// TIA Portal V17 export
// export: Created 2022-07-20T07:01:25.3960544Z, ExportSetting WithDefaults, DisplayName Totally Integrated Automation Portal, DisplayVersion V17, DisplayName TIA Portal Openness, DisplayVersion V17, DisplayName TIA Portal Version Control Interface, DisplayVersion V17, DisplayName SINAMICS Startdrive Advanced, DisplayVersion V17, DisplayName SINAMICS Startdrive G130, G150, S120, S150, SINAMICS MV, S210, DisplayVersion V17, DisplayName SINAMICS Startdrive G110M, G120, G120C, G120D, G120P, G115D, DisplayVersion V17, DisplayName STEP 7 Professional, DisplayVersion V17, DisplayName STEP 7 Safety, DisplayVersion V17, DisplayName WinCC Advanced, DisplayVersion V17
FUNCTION_BLOCK "FB10230_LAM_LexiumDriver"   // FB10230, LAD
{ S7_Optimized_Access := 'TRUE' }
AUTHOR : Schneider_Electric
FAMILY : Lexium_MDrive
VERSION : 1.0
// stored: AutoNumber false, IsIECCheckEnabled false, IsRetainMemResEnabled false, MemoryReserve 100, SetENOAutomatically false, UDAEnableTagReadback false
   VAR_INPUT
      Drive_In : "TLexium_MDrv_Drv2Plc";
      UseInputsOutputs : Bool;
      Move_Type : DInt;
      Home_Type : SInt := 1;
      Position : DInt;
      Speed : DWord := 20000;
      Jog_Speed : DInt := 75000;
      Accel_Rate : DWord := 10000;
      Decel_Rate : DWord := 10000;
      Initial_Vel : DWord := 1000;
      Hold_Current : SInt := 5;
      Run_Current : SInt := 25;
      MicrostepValue : DInt := 256;
      Enable : Bool;
      Start : Bool;
      Stop : Bool;
      Jog_Fwd : Bool;
      Jog_Rev : Bool;
      Acknowledge : Bool;
      Home : Bool;
      Zero_Home_Pos : Bool := false;
      Out1_Set : Bool;
      Out2_Set : Bool;
      Out3_Set : Bool;
   END_VAR
   VAR_OUTPUT
      Drive_Out : "TLexium_MDrv_Plc2Drv";
      Pos_Fdbk : DInt;
      Error_Code : UInt;
      DN : Bool;
      ER : Bool;
      IP : Bool;
      In1 : Bool;
      In2 : Bool;
      In3 : Bool;
      In4 : Bool;
   END_VAR
   VAR
      Jog_Perm : Bool;
      Jog_Fwd_Req : Bool;
      Jog_Rev_Req : Bool;
      Stop_Act : Bool;
      Abs_Act : Bool;
      Rel_Act : Bool;
      HM_Act : Bool;
      Start_OS : Bool;
      MV_Stop_OS : Bool;
      Set_Pos_Zero : Bool;
      Slew_Rate : DInt;
      Slew_Rate_Prev : DInt;
      MicrostepValue_Prev : DInt;
      SetAccTmr { S7_SetPoint := 'True'} : TOF_TIME;
      SetDecTmr { S7_SetPoint := 'True'} : TOF_TIME;
      SetTSTmr { S7_SetPoint := 'True'} : TOF_TIME;
      SetVITmr { S7_SetPoint := 'True'} : TOF_TIME;
      SetVMTmr { S7_SetPoint := 'True'} : TOF_TIME;
      SetHCTmr { S7_SetPoint := 'True'} : TOF_TIME;
      SetRCTmr { S7_SetPoint := 'True'} : TOF_TIME;
      SetTQTmr { S7_SetPoint := 'True'} : TOF_TIME;
      SetSLTmr { S7_SetPoint := 'True'} : TOF_TIME;
      ABS_Tmr { S7_SetPoint := 'True'} : TOF_TIME;
      REL_Tmr { S7_SetPoint := 'True'} : TOF_TIME;
      HM_Tmr { S7_SetPoint := 'True'} : TOF_TIME;
      MS_Tmr { S7_SetPoint := 'True'} : TOF_TIME;
      SetZero_Tmr { S7_SetPoint := 'True'} : TOF_TIME;
      ClrErr_Tmr { S7_SetPoint := 'True'} : TOF_TIME;
      Stop_Dly_Tmr { S7_SetPoint := 'True'} : TON_TIME;
      ACC_PMem : Bool;
      DEC_PMem : Bool;
      TS_PMem : Bool;
      VI_PMem : Bool;
      VM_PMem : Bool;
      HC_PMem : Bool;
      RC_PMem : Bool;
      TQ_PMem : Bool;
      SL_PMem : Bool;
      MS_Pmem : Bool;
      Start_PMem : Bool;
      MV_NMem : Bool;
      ABS_PMem : Bool;
      REL_PMem : Bool;
      HM_PMem : Bool;
      Set_Zero_PMem : Bool;
      ClrErr_PMem : Bool;
      AckErr_Pmem : Bool;
      Stop_PMem : Bool;
      MV_Stop_Tmr { S7_SetPoint := 'True'} : TON_TIME;
      IS_PMem { S7_SetPoint := 'True'} : Bool;
      FB10232_Lam_WriteISMessages_Instance { S7_SetPoint := 'True'} : "FB10232_LAM_WriteISMessages";
   END_VAR
   VAR_TEMP
      Inputs : SInt;
      Hold_Cur_SP : SInt;
      Run_Cur_SP : SInt;
      Torque_SP : SInt;
      Move_Type_Loc : DInt;
      Home_Type_Loc : SInt;
      Position_SP : DInt;
      _SetAccTmr_ET : Time;
      _SetDecTmr_ET : Time;
      _SetTSTmr_ET : Time;
      _SetVITmr_ET : Time;
      _SetVMTmr_ET : Time;
      _SetHCTmr_ET : Time;
      _SetRCTmr_ET : Time;
      _SetTQTmr_ET : Time;
      _SetSLTmr_ET : Time;
      _Abs_Tmr_ET : Time;
      _Rel_Tmr_ET : Time;
      _HM_Tmr_ET : Time;
      _SetZero_Tmr_ET : Time;
      _Stop_Dly_Tmr_ET : Time;
      _ClrErr_Tmr_ET : Time;
      Outputs : SInt;
   END_VAR
   // Drive_Out.AS := 2;   // 2 = Mode hybride
   VAR_TEMP   // added for the SCL form of the ladder/FBD networks
      _w1 : Bool;
      _w2 : Bool;
      _w3 : Bool;
      _w4 : Bool;
   END_VAR
BEGIN

REGION Network 1: States of Inputs In1, 2, 3, 4
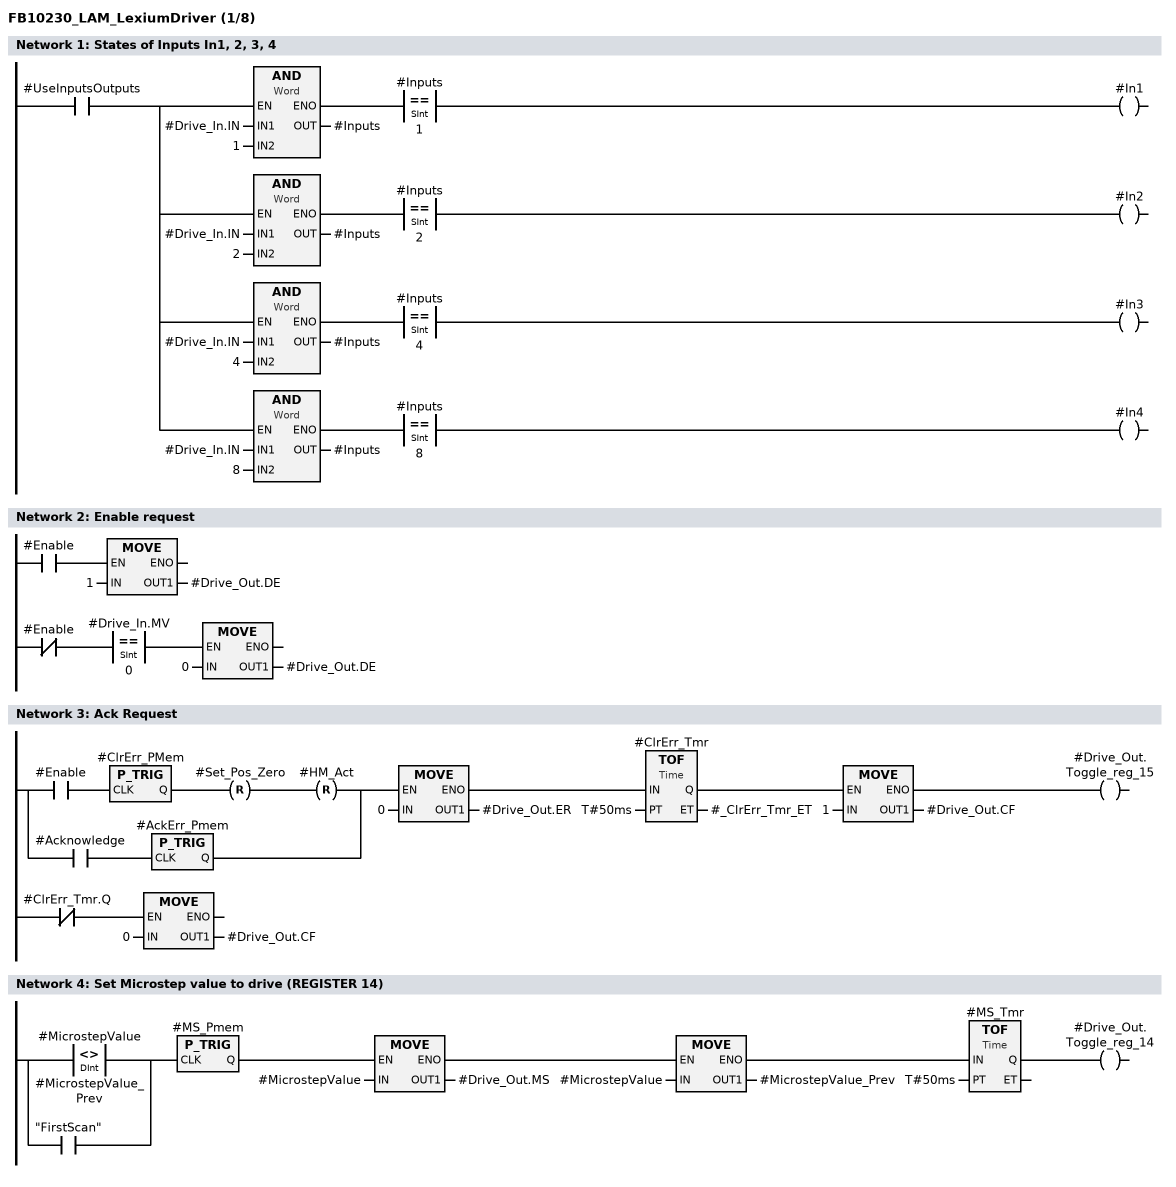
   RUNG wire#powerrail
      Contact( #UseInputsOutputs )
      wire#w1
      { S7_Templates := "SrcType := Word" } And(in1 := #Drive_In.IN, in2 := 1, out => #Inputs)
      { S7_Templates := "SrcType := SInt" } EQ_Contact(in1 := #Inputs, in2 := 1)
      Coil( #In1 )
   END_RUNG
   RUNG wire#w1
      { S7_Templates := "SrcType := Word" } And(in1 := #Drive_In.IN, in2 := 2, out => #Inputs)
      { S7_Templates := "SrcType := SInt" } EQ_Contact(in1 := #Inputs, in2 := 2)
      Coil( #In2 )
   END_RUNG
   RUNG wire#w1
      { S7_Templates := "SrcType := Word" } And(in1 := #Drive_In.IN, in2 := 4, out => #Inputs)
      { S7_Templates := "SrcType := SInt" } EQ_Contact(in1 := #Inputs, in2 := 4)
      Coil( #In3 )
   END_RUNG
   RUNG wire#w1
      { S7_Templates := "SrcType := Word" } And(in1 := #Drive_In.IN, in2 := 8, out => #Inputs)
      { S7_Templates := "SrcType := SInt" } EQ_Contact(in1 := #Inputs, in2 := 8)
      Coil( #In4 )
   END_RUNG
   // the same network as SCL:
   IF #UseInputsOutputs THEN #Inputs := #Drive_In.IN AND 1; END_IF;
   #In1 := #UseInputsOutputs AND (#Inputs = 1);
   IF #UseInputsOutputs THEN #Inputs := #Drive_In.IN AND 2; END_IF;
   #In2 := #UseInputsOutputs AND (#Inputs = 2);
   IF #UseInputsOutputs THEN #Inputs := #Drive_In.IN AND 4; END_IF;
   #In3 := #UseInputsOutputs AND (#Inputs = 4);
   IF #UseInputsOutputs THEN #Inputs := #Drive_In.IN AND 8; END_IF;
   #In4 := #UseInputsOutputs AND (#Inputs = 8);
END_REGION

REGION Network 2: Enable request
   RUNG wire#powerrail
      Contact( #Enable )
      Move(in := 1, out1 => #Drive_Out.DE)
   END_RUNG
   RUNG wire#powerrail
      I_Contact( #Enable )
      { S7_Templates := "SrcType := SInt" } EQ_Contact(in1 := #Drive_In.MV, in2 := 0)
      Move(in := 0, out1 => #Drive_Out.DE)
   END_RUNG
   // the same network as SCL:
   IF #Enable THEN #Drive_Out.DE := 1; END_IF;
   IF NOT #Enable AND (#Drive_In.MV = 0) THEN #Drive_Out.DE := 0; END_IF;
END_REGION

REGION Network 3: Ack Request
   RUNG wire#powerrail
      Contact( #Enable )
      P_Trig( #ClrErr_PMem )
      R_Coil( #Set_Pos_Zero )
      R_Coil( #HM_Act )
      wire#w1
      Move(in := 0, out1 => #Drive_Out.ER)
      { S7_Templates := "time_type := Time" } #ClrErr_Tmr.TOF(pt := T#50ms, et => #_ClrErr_Tmr_ET)
      Move(in := 1, out1 => #Drive_Out.CF)
      Coil( #Drive_Out.Toggle_reg_15 )
   END_RUNG
   RUNG wire#powerrail
      Contact( #Acknowledge )
      P_Trig( #AckErr_Pmem )
   END_RUNG wire#w1
   RUNG wire#powerrail
      I_Contact( #ClrErr_Tmr.Q )
      Move(in := 0, out1 => #Drive_Out.CF)
   END_RUNG
   // the same network as SCL:
   #_w1 := #Enable AND NOT #ClrErr_PMem;   // rising edge
   #ClrErr_PMem := #Enable;
   IF #_w1 THEN
       #Set_Pos_Zero := FALSE;
       #HM_Act := FALSE;
   END_IF;
   #_w2 := #Acknowledge AND NOT #AckErr_Pmem;   // rising edge
   #AckErr_Pmem := #Acknowledge;
   #_w3 := #_w1 OR #_w2;
   IF #_w3 THEN #Drive_Out.ER := 0; END_IF;
   #ClrErr_Tmr(IN := #_w3, PT := T#50ms, ET => #_ClrErr_Tmr_ET);   // TOF
   IF #ClrErr_Tmr.Q THEN #Drive_Out.CF := 1; END_IF;
   #Drive_Out.Toggle_reg_15 := #ClrErr_Tmr.Q;
   IF NOT #ClrErr_Tmr.Q THEN #Drive_Out.CF := 0; END_IF;
END_REGION

REGION Network 4: Set Microstep value to drive (REGISTER 14)
   RUNG wire#powerrail
      { S7_Templates := "SrcType := DInt" } NE_Contact(in1 := #MicrostepValue, in2 := #MicrostepValue_Prev)
      wire#w1
      P_Trig( #MS_Pmem )
      Move(in := #MicrostepValue, out1 => #Drive_Out.MS)
      Move(in := #MicrostepValue, out1 => #MicrostepValue_Prev)
      { S7_Templates := "time_type := Time" } #MS_Tmr.TOF(pt := T#50ms, et =>)
      Coil( #Drive_Out.Toggle_reg_14 )
   END_RUNG
   RUNG wire#powerrail
      Contact( "FirstScan" )
   END_RUNG wire#w1
   // the same network as SCL:
   #_w1 := (#MicrostepValue <> #MicrostepValue_Prev) OR "FirstScan";
   #_w2 := #_w1 AND NOT #MS_Pmem;   // rising edge
   #MS_Pmem := #_w1;
   IF #_w2 THEN
       #Drive_Out.MS := #MicrostepValue;
       #MicrostepValue_Prev := #MicrostepValue;
   END_IF;
   #MS_Tmr(IN := #_w2, PT := T#50ms);   // TOF
   #Drive_Out.Toggle_reg_14 := #MS_Tmr.Q;
END_REGION

REGION Network 5: Hold Current limits
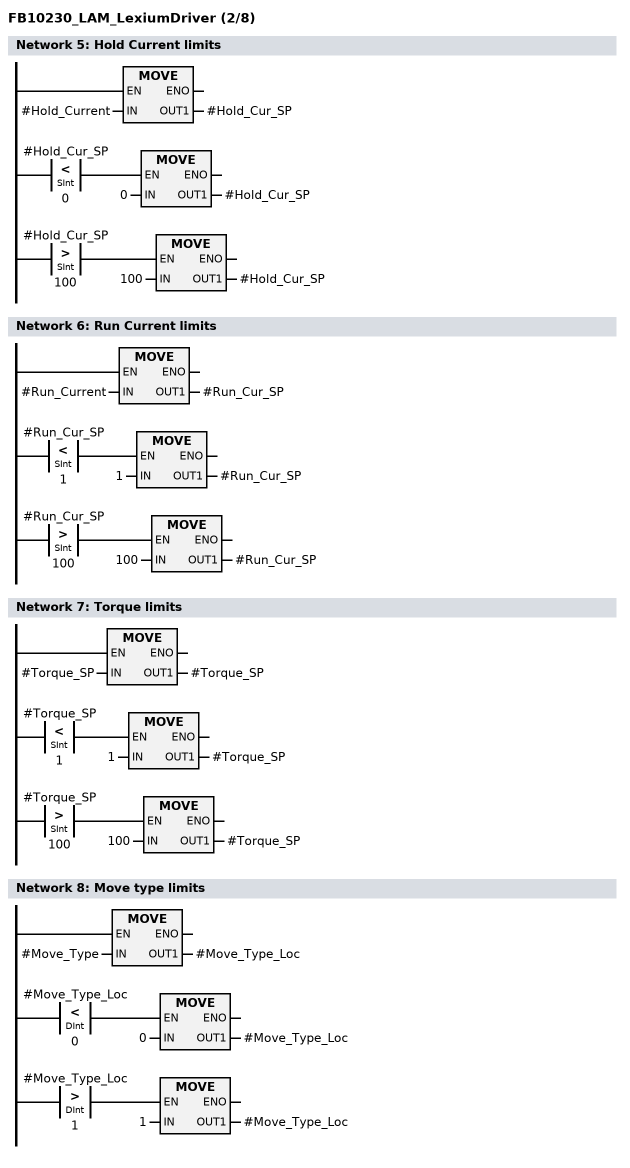
   RUNG wire#powerrail
      Move(in := #Hold_Current, out1 => #Hold_Cur_SP)
   END_RUNG
   RUNG wire#powerrail
      { S7_Templates := "SrcType := SInt" } LT_Contact(in1 := #Hold_Cur_SP, in2 := 0)
      Move(in := 0, out1 => #Hold_Cur_SP)
   END_RUNG
   RUNG wire#powerrail
      { S7_Templates := "SrcType := SInt" } GT_Contact(in1 := #Hold_Cur_SP, in2 := 100)
      Move(in := 100, out1 => #Hold_Cur_SP)
   END_RUNG
   // the same network as SCL:
   #Hold_Cur_SP := #Hold_Current;
   IF #Hold_Cur_SP < 0 THEN #Hold_Cur_SP := 0; END_IF;
   IF #Hold_Cur_SP > 100 THEN #Hold_Cur_SP := 100; END_IF;
END_REGION

REGION Network 6: Run Current limits
   RUNG wire#powerrail
      Move(in := #Run_Current, out1 => #Run_Cur_SP)
   END_RUNG
   RUNG wire#powerrail
      { S7_Templates := "SrcType := SInt" } LT_Contact(in1 := #Run_Cur_SP, in2 := 1)
      Move(in := 1, out1 => #Run_Cur_SP)
   END_RUNG
   RUNG wire#powerrail
      { S7_Templates := "SrcType := SInt" } GT_Contact(in1 := #Run_Cur_SP, in2 := 100)
      Move(in := 100, out1 => #Run_Cur_SP)
   END_RUNG
   // the same network as SCL:
   #Run_Cur_SP := #Run_Current;
   IF #Run_Cur_SP < 1 THEN #Run_Cur_SP := 1; END_IF;
   IF #Run_Cur_SP > 100 THEN #Run_Cur_SP := 100; END_IF;
END_REGION

REGION Network 7: Torque limits
   RUNG wire#powerrail
      Move(in := #Torque_SP, out1 => #Torque_SP)
   END_RUNG
   RUNG wire#powerrail
      { S7_Templates := "SrcType := SInt" } LT_Contact(in1 := #Torque_SP, in2 := 1)
      Move(in := 1, out1 => #Torque_SP)
   END_RUNG
   RUNG wire#powerrail
      { S7_Templates := "SrcType := SInt" } GT_Contact(in1 := #Torque_SP, in2 := 100)
      Move(in := 100, out1 => #Torque_SP)
   END_RUNG
   // the same network as SCL:
   #Torque_SP := #Torque_SP;
   IF #Torque_SP < 1 THEN #Torque_SP := 1; END_IF;
   IF #Torque_SP > 100 THEN #Torque_SP := 100; END_IF;
END_REGION

REGION Network 8: Move type limits
   RUNG wire#powerrail
      Move(in := #Move_Type, out1 => #Move_Type_Loc)
   END_RUNG
   RUNG wire#powerrail
      { S7_Templates := "SrcType := DInt" } LT_Contact(in1 := #Move_Type_Loc, in2 := 0)
      Move(in := 0, out1 => #Move_Type_Loc)
   END_RUNG
   RUNG wire#powerrail
      { S7_Templates := "SrcType := DInt" } GT_Contact(in1 := #Move_Type_Loc, in2 := 1)
      Move(in := 1, out1 => #Move_Type_Loc)
   END_RUNG
   // the same network as SCL:
   #Move_Type_Loc := #Move_Type;
   IF #Move_Type_Loc < 0 THEN #Move_Type_Loc := 0; END_IF;
   IF #Move_Type_Loc > 1 THEN #Move_Type_Loc := 1; END_IF;
END_REGION

REGION Network 9: Home type limits
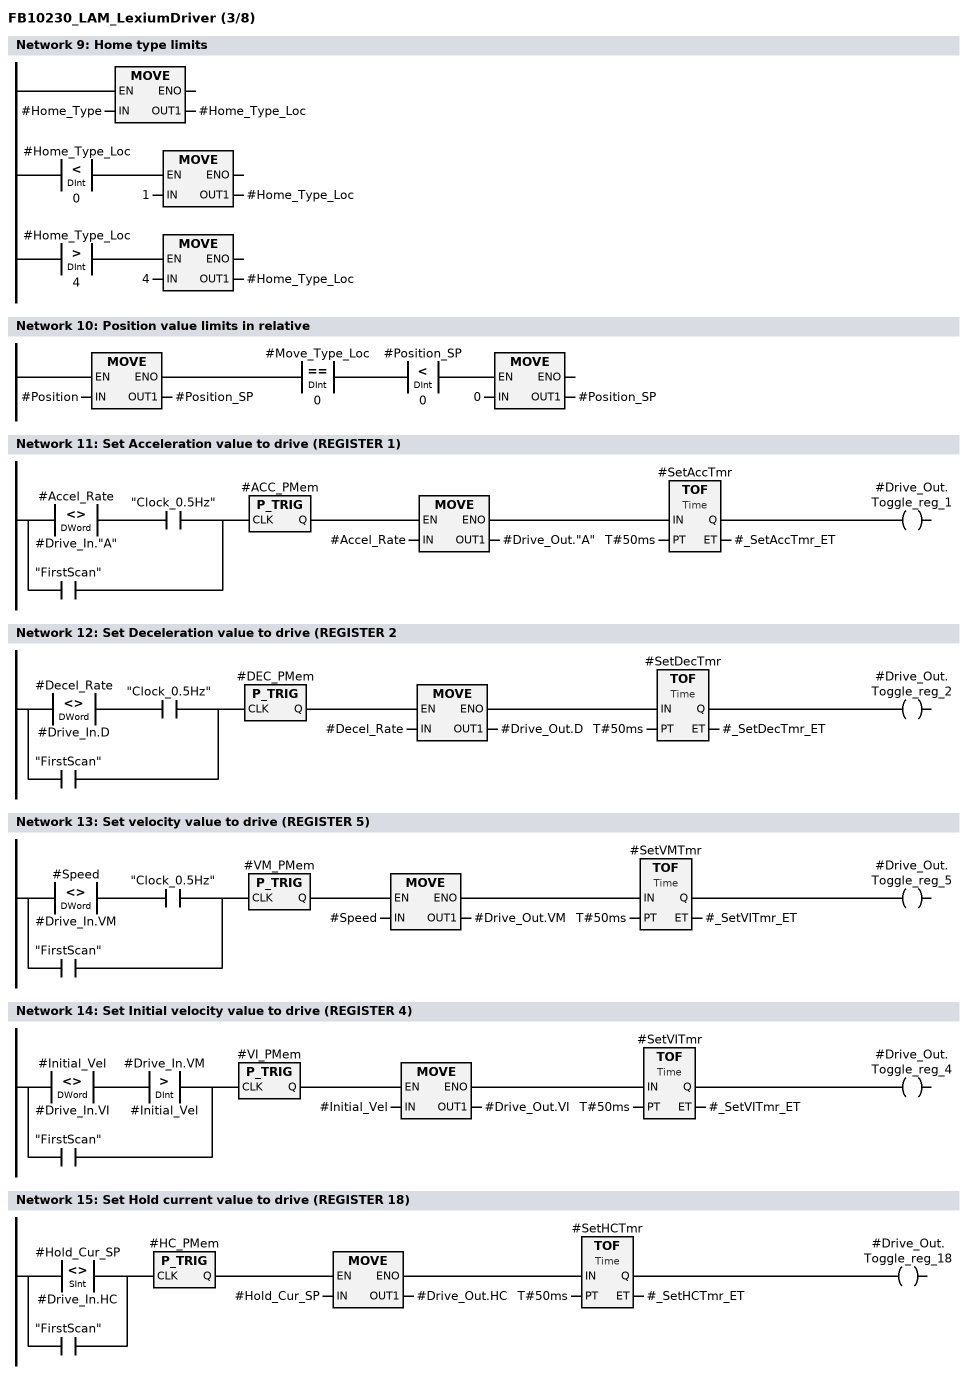
   RUNG wire#powerrail
      Move(in := #Home_Type, out1 => #Home_Type_Loc)
   END_RUNG
   RUNG wire#powerrail
      { S7_Templates := "SrcType := DInt" } LT_Contact(in1 := #Home_Type_Loc, in2 := 0)
      Move(in := 1, out1 => #Home_Type_Loc)
   END_RUNG
   RUNG wire#powerrail
      { S7_Templates := "SrcType := DInt" } GT_Contact(in1 := #Home_Type_Loc, in2 := 4)
      Move(in := 4, out1 => #Home_Type_Loc)
   END_RUNG
   // the same network as SCL:
   #Home_Type_Loc := #Home_Type;
   IF #Home_Type_Loc < 0 THEN #Home_Type_Loc := 1; END_IF;
   IF #Home_Type_Loc > 4 THEN #Home_Type_Loc := 4; END_IF;
END_REGION

REGION Network 10: Position value limits in relative
   RUNG wire#powerrail
      Move(in := #Position, out1 => #Position_SP)
      { S7_Templates := "SrcType := DInt" } EQ_Contact(in1 := #Move_Type_Loc, in2 := 0)
      { S7_Templates := "SrcType := DInt" } LT_Contact(in1 := #Position_SP, in2 := 0)
      Move(in := 0, out1 => #Position_SP)
   END_RUNG
   // the same network as SCL:
   #Position_SP := #Position;
   IF (#Move_Type_Loc = 0) AND (#Position_SP < 0) THEN #Position_SP := 0; END_IF;
END_REGION

REGION Network 11: Set Acceleration value to drive (REGISTER 1)
   RUNG wire#powerrail
      { S7_Templates := "SrcType := DWord" } NE_Contact(in1 := #Accel_Rate, in2 := #Drive_In."A")
      Contact( "Clock_0.5Hz" )
      wire#w1
      P_Trig( #ACC_PMem )
      Move(in := #Accel_Rate, out1 => #Drive_Out."A")
      { S7_Templates := "time_type := Time" } #SetAccTmr.TOF(pt := T#50ms, et => #_SetAccTmr_ET)
      Coil( #Drive_Out.Toggle_reg_1 )
   END_RUNG
   RUNG wire#powerrail
      Contact( "FirstScan" )
   END_RUNG wire#w1
   // the same network as SCL:
   #_w1 := ((#Accel_Rate <> #Drive_In."A") AND "Clock_0.5Hz") OR "FirstScan";
   #_w2 := #_w1 AND NOT #ACC_PMem;   // rising edge
   #ACC_PMem := #_w1;
   IF #_w2 THEN #Drive_Out."A" := #Accel_Rate; END_IF;
   #SetAccTmr(IN := #_w2, PT := T#50ms, ET => #_SetAccTmr_ET);   // TOF
   #Drive_Out.Toggle_reg_1 := #SetAccTmr.Q;
END_REGION

REGION Network 12: Set Deceleration value to drive (REGISTER 2
   RUNG wire#powerrail
      { S7_Templates := "SrcType := DWord" } NE_Contact(in1 := #Decel_Rate, in2 := #Drive_In.D)
      Contact( "Clock_0.5Hz" )
      wire#w1
      P_Trig( #DEC_PMem )
      Move(in := #Decel_Rate, out1 => #Drive_Out.D)
      { S7_Templates := "time_type := Time" } #SetDecTmr.TOF(pt := T#50ms, et => #_SetDecTmr_ET)
      Coil( #Drive_Out.Toggle_reg_2 )
   END_RUNG
   RUNG wire#powerrail
      Contact( "FirstScan" )
   END_RUNG wire#w1
   // the same network as SCL:
   #_w1 := ((#Decel_Rate <> #Drive_In.D) AND "Clock_0.5Hz") OR "FirstScan";
   #_w2 := #_w1 AND NOT #DEC_PMem;   // rising edge
   #DEC_PMem := #_w1;
   IF #_w2 THEN #Drive_Out.D := #Decel_Rate; END_IF;
   #SetDecTmr(IN := #_w2, PT := T#50ms, ET => #_SetDecTmr_ET);   // TOF
   #Drive_Out.Toggle_reg_2 := #SetDecTmr.Q;
END_REGION

REGION Network 13: Set velocity value to drive (REGISTER 5)
   RUNG wire#powerrail
      { S7_Templates := "SrcType := DWord" } NE_Contact(in1 := #Speed, in2 := #Drive_In.VM)
      Contact( "Clock_0.5Hz" )
      wire#w1
      P_Trig( #VM_PMem )
      Move(in := #Speed, out1 => #Drive_Out.VM)
      { S7_Templates := "time_type := Time" } #SetVMTmr.TOF(pt := T#50ms, et => #_SetVITmr_ET)
      Coil( #Drive_Out.Toggle_reg_5 )
   END_RUNG
   RUNG wire#powerrail
      Contact( "FirstScan" )
   END_RUNG wire#w1
   // the same network as SCL:
   #_w1 := ((#Speed <> #Drive_In.VM) AND "Clock_0.5Hz") OR "FirstScan";
   #_w2 := #_w1 AND NOT #VM_PMem;   // rising edge
   #VM_PMem := #_w1;
   IF #_w2 THEN #Drive_Out.VM := #Speed; END_IF;
   #SetVMTmr(IN := #_w2, PT := T#50ms, ET => #_SetVITmr_ET);   // TOF
   #Drive_Out.Toggle_reg_5 := #SetVMTmr.Q;
END_REGION

REGION Network 14: Set Initial velocity value to drive (REGISTER 4)
   RUNG wire#powerrail
      { S7_Templates := "SrcType := DWord" } NE_Contact(in1 := #Initial_Vel, in2 := #Drive_In.VI)
      { S7_Templates := "SrcType := DInt" } GT_Contact(in1 := #Drive_In.VM, in2 := #Initial_Vel)
      wire#w1
      P_Trig( #VI_PMem )
      Move(in := #Initial_Vel, out1 => #Drive_Out.VI)
      { S7_Templates := "time_type := Time" } #SetVITmr.TOF(pt := T#50ms, et => #_SetVITmr_ET)
      Coil( #Drive_Out.Toggle_reg_4 )
   END_RUNG
   RUNG wire#powerrail
      Contact( "FirstScan" )
   END_RUNG wire#w1
   // the same network as SCL:
   #_w1 := ((#Initial_Vel <> #Drive_In.VI) AND (#Drive_In.VM > #Initial_Vel)) OR "FirstScan";
   #_w2 := #_w1 AND NOT #VI_PMem;   // rising edge
   #VI_PMem := #_w1;
   IF #_w2 THEN #Drive_Out.VI := #Initial_Vel; END_IF;
   #SetVITmr(IN := #_w2, PT := T#50ms, ET => #_SetVITmr_ET);   // TOF
   #Drive_Out.Toggle_reg_4 := #SetVITmr.Q;
END_REGION

REGION Network 15: Set Hold current value to drive (REGISTER 18)
   RUNG wire#powerrail
      { S7_Templates := "SrcType := SInt" } NE_Contact(in1 := #Hold_Cur_SP, in2 := #Drive_In.HC)
      wire#w1
      P_Trig( #HC_PMem )
      Move(in := #Hold_Cur_SP, out1 => #Drive_Out.HC)
      { S7_Templates := "time_type := Time" } #SetHCTmr.TOF(pt := T#50ms, et => #_SetHCTmr_ET)
      Coil( #Drive_Out.Toggle_reg_18 )
   END_RUNG
   RUNG wire#powerrail
      Contact( "FirstScan" )
   END_RUNG wire#w1
   // the same network as SCL:
   #_w1 := (#Hold_Cur_SP <> #Drive_In.HC) OR "FirstScan";
   #_w2 := #_w1 AND NOT #HC_PMem;   // rising edge
   #HC_PMem := #_w1;
   IF #_w2 THEN #Drive_Out.HC := #Hold_Cur_SP; END_IF;
   #SetHCTmr(IN := #_w2, PT := T#50ms, ET => #_SetHCTmr_ET);   // TOF
   #Drive_Out.Toggle_reg_18 := #SetHCTmr.Q;
END_REGION

REGION Network 16: Set Run current value to drive (REGISTER 20)
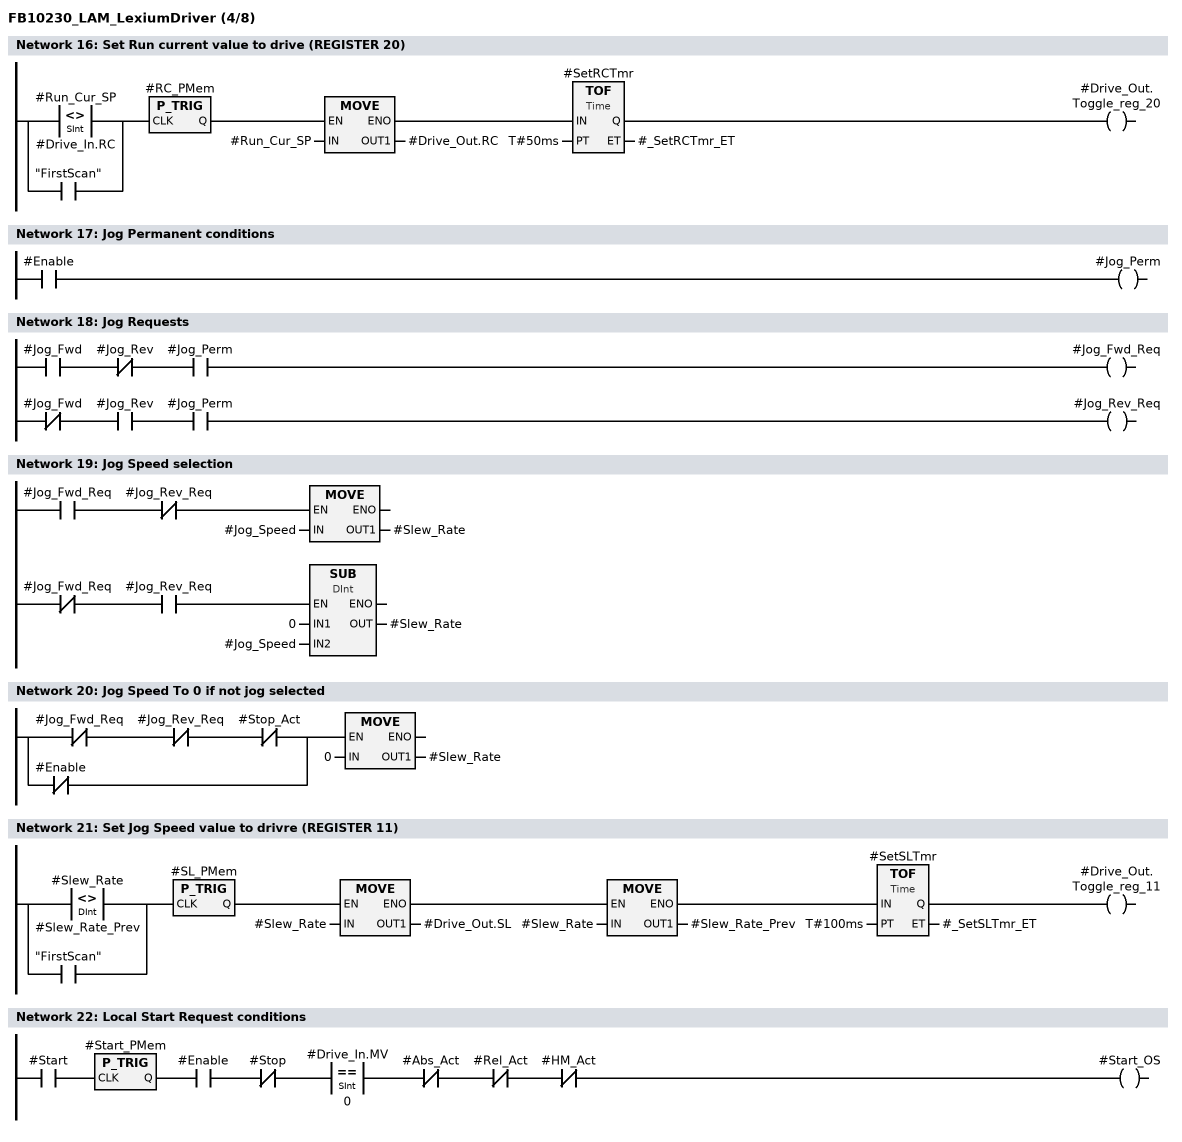
   RUNG wire#powerrail
      { S7_Templates := "SrcType := SInt" } NE_Contact(in1 := #Run_Cur_SP, in2 := #Drive_In.RC)
      wire#w1
      P_Trig( #RC_PMem )
      Move(in := #Run_Cur_SP, out1 => #Drive_Out.RC)
      { S7_Templates := "time_type := Time" } #SetRCTmr.TOF(pt := T#50ms, et => #_SetRCTmr_ET)
      Coil( #Drive_Out.Toggle_reg_20 )
   END_RUNG
   RUNG wire#powerrail
      Contact( "FirstScan" )
   END_RUNG wire#w1
   // the same network as SCL:
   #_w1 := (#Run_Cur_SP <> #Drive_In.RC) OR "FirstScan";
   #_w2 := #_w1 AND NOT #RC_PMem;   // rising edge
   #RC_PMem := #_w1;
   IF #_w2 THEN #Drive_Out.RC := #Run_Cur_SP; END_IF;
   #SetRCTmr(IN := #_w2, PT := T#50ms, ET => #_SetRCTmr_ET);   // TOF
   #Drive_Out.Toggle_reg_20 := #SetRCTmr.Q;
END_REGION

REGION Network 17: Jog Permanent conditions
   RUNG wire#powerrail
      Contact( #Enable )
      Coil( #Jog_Perm )
   END_RUNG
   // the same network as SCL:
   #Jog_Perm := #Enable;
END_REGION

REGION Network 18: Jog Requests
   RUNG wire#powerrail
      Contact( #Jog_Fwd )
      I_Contact( #Jog_Rev )
      Contact( #Jog_Perm )
      Coil( #Jog_Fwd_Req )
   END_RUNG
   RUNG wire#powerrail
      I_Contact( #Jog_Fwd )
      Contact( #Jog_Rev )
      Contact( #Jog_Perm )
      Coil( #Jog_Rev_Req )
   END_RUNG
   // the same network as SCL:
   #Jog_Fwd_Req := #Jog_Fwd AND NOT #Jog_Rev AND #Jog_Perm;
   #Jog_Rev_Req := NOT #Jog_Fwd AND #Jog_Rev AND #Jog_Perm;
END_REGION

REGION Network 19: Jog Speed selection
   RUNG wire#powerrail
      Contact( #Jog_Fwd_Req )
      I_Contact( #Jog_Rev_Req )
      Move(in := #Jog_Speed, out1 => #Slew_Rate)
   END_RUNG
   RUNG wire#powerrail
      I_Contact( #Jog_Fwd_Req )
      Contact( #Jog_Rev_Req )
      { S7_Templates := "SrcType := DInt" } Sub(in1 := 0, in2 := #Jog_Speed, out => #Slew_Rate)
   END_RUNG
   // the same network as SCL:
   IF #Jog_Fwd_Req AND NOT #Jog_Rev_Req THEN #Slew_Rate := #Jog_Speed; END_IF;
   IF NOT #Jog_Fwd_Req AND #Jog_Rev_Req THEN #Slew_Rate := 0 - #Jog_Speed; END_IF;
END_REGION

REGION Network 20: Jog Speed To 0 if not jog selected
   RUNG wire#powerrail
      I_Contact( #Jog_Fwd_Req )
      I_Contact( #Jog_Rev_Req )
      I_Contact( #Stop_Act )
      wire#w1
      Move(in := 0, out1 => #Slew_Rate)
   END_RUNG
   RUNG wire#powerrail
      I_Contact( #Enable )
   END_RUNG wire#w1
   // the same network as SCL:
   IF (NOT #Jog_Fwd_Req AND NOT #Jog_Rev_Req AND NOT #Stop_Act) OR NOT #Enable THEN #Slew_Rate := 0; END_IF;
END_REGION

REGION Network 21: Set Jog Speed value to drivre (REGISTER 11)
   RUNG wire#powerrail
      { S7_Templates := "SrcType := DInt" } NE_Contact(in1 := #Slew_Rate, in2 := #Slew_Rate_Prev)
      wire#w1
      P_Trig( #SL_PMem )
      Move(in := #Slew_Rate, out1 => #Drive_Out.SL)
      Move(in := #Slew_Rate, out1 => #Slew_Rate_Prev)
      { S7_Templates := "time_type := Time" } #SetSLTmr.TOF(pt := T#100ms, et => #_SetSLTmr_ET)
      Coil( #Drive_Out.Toggle_reg_11 )
   END_RUNG
   RUNG wire#powerrail
      Contact( "FirstScan" )
   END_RUNG wire#w1
   // the same network as SCL:
   #_w1 := (#Slew_Rate <> #Slew_Rate_Prev) OR "FirstScan";
   #_w2 := #_w1 AND NOT #SL_PMem;   // rising edge
   #SL_PMem := #_w1;
   IF #_w2 THEN
       #Drive_Out.SL := #Slew_Rate;
       #Slew_Rate_Prev := #Slew_Rate;
   END_IF;
   #SetSLTmr(IN := #_w2, PT := T#100ms, ET => #_SetSLTmr_ET);   // TOF
   #Drive_Out.Toggle_reg_11 := #SetSLTmr.Q;
END_REGION

REGION Network 22: Local Start Request conditions
   RUNG wire#powerrail
      Contact( #Start )
      P_Trig( #Start_PMem )
      Contact( #Enable )
      I_Contact( #Stop )
      { S7_Templates := "SrcType := SInt" } EQ_Contact(in1 := #Drive_In.MV, in2 := 0)
      I_Contact( #Abs_Act )
      I_Contact( #Rel_Act )
      I_Contact( #HM_Act )
      Coil( #Start_OS )
   END_RUNG
   // the same network as SCL:
   #_w1 := #Start AND NOT #Start_PMem;   // rising edge
   #Start_PMem := #Start;
   #Start_OS := #_w1 AND #Enable AND NOT #Stop AND (#Drive_In.MV = 0) AND NOT #Abs_Act AND NOT #Rel_Act AND NOT #HM_Act;
END_REGION

REGION Network 23: Local Stop state
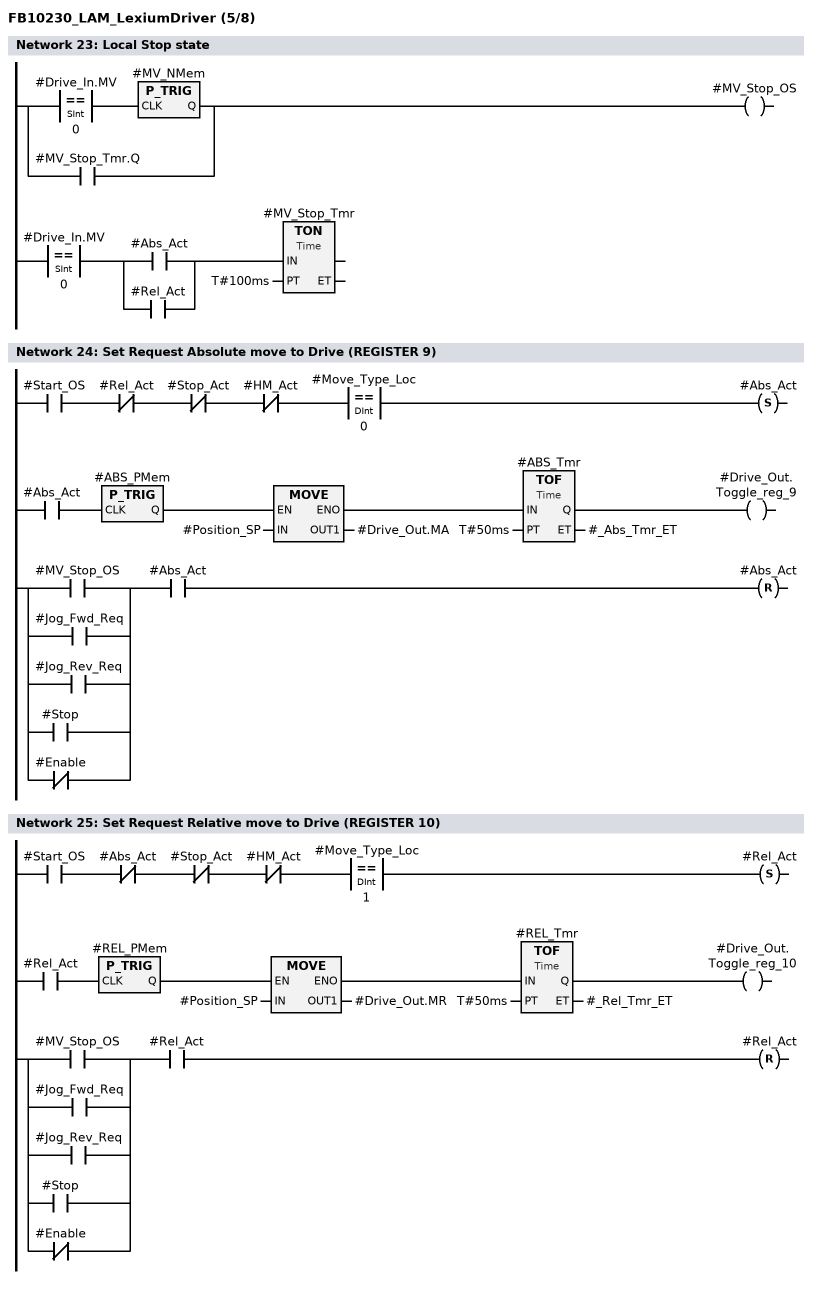
   RUNG wire#powerrail
      { S7_Templates := "SrcType := SInt" } EQ_Contact(in1 := #Drive_In.MV, in2 := 0)
      P_Trig( #MV_NMem )
      wire#w1
      Coil( #MV_Stop_OS )
   END_RUNG
   RUNG wire#powerrail
      Contact( #MV_Stop_Tmr.Q )
   END_RUNG wire#w1
   RUNG wire#powerrail
      { S7_Templates := "SrcType := SInt" } EQ_Contact(in1 := #Drive_In.MV, in2 := 0)
      wire#w2
      Contact( #Abs_Act )
      wire#w3
      { S7_Templates := "time_type := Time" } #MV_Stop_Tmr.TON(pt := T#100ms, et =>)
   END_RUNG
   RUNG wire#w2
      Contact( #Rel_Act )
   END_RUNG wire#w3
   // the same network as SCL:
   #_w1 := #Drive_In.MV = 0;
   #_w2 := #_w1 AND NOT #MV_NMem;   // rising edge
   #MV_NMem := #_w1;
   #MV_Stop_OS := #_w2 OR #MV_Stop_Tmr.Q;
   #MV_Stop_Tmr(IN := (#Drive_In.MV = 0) AND (#Abs_Act OR #Rel_Act), PT := T#100ms);   // TON
END_REGION

REGION Network 24: Set Request Absolute move to Drive (REGISTER 9)
   RUNG wire#powerrail
      Contact( #Start_OS )
      I_Contact( #Rel_Act )
      I_Contact( #Stop_Act )
      I_Contact( #HM_Act )
      { S7_Templates := "SrcType := DInt" } EQ_Contact(in1 := #Move_Type_Loc, in2 := 0)
      S_Coil( #Abs_Act )
   END_RUNG
   RUNG wire#powerrail
      Contact( #Abs_Act )
      P_Trig( #ABS_PMem )
      Move(in := #Position_SP, out1 => #Drive_Out.MA)
      { S7_Templates := "time_type := Time" } #ABS_Tmr.TOF(pt := T#50ms, et => #_Abs_Tmr_ET)
      Coil( #Drive_Out.Toggle_reg_9 )
   END_RUNG
   RUNG wire#powerrail
      Contact( #MV_Stop_OS )
      wire#w1
      Contact( #Abs_Act )
      R_Coil( #Abs_Act )
   END_RUNG
   RUNG wire#powerrail
      Contact( #Jog_Fwd_Req )
   END_RUNG wire#w1
   RUNG wire#powerrail
      Contact( #Jog_Rev_Req )
   END_RUNG wire#w1
   RUNG wire#powerrail
      Contact( #Stop )
   END_RUNG wire#w1
   RUNG wire#powerrail
      I_Contact( #Enable )
   END_RUNG wire#w1
   // the same network as SCL:
   IF #Start_OS AND NOT #Rel_Act AND NOT #Stop_Act AND NOT #HM_Act AND (#Move_Type_Loc = 0) THEN
       #Abs_Act := TRUE;
   END_IF;
   #_w1 := #Abs_Act AND NOT #ABS_PMem;   // rising edge
   #ABS_PMem := #Abs_Act;
   IF #_w1 THEN #Drive_Out.MA := #Position_SP; END_IF;
   #ABS_Tmr(IN := #_w1, PT := T#50ms, ET => #_Abs_Tmr_ET);   // TOF
   #Drive_Out.Toggle_reg_9 := #ABS_Tmr.Q;
   IF (#MV_Stop_OS OR #Jog_Fwd_Req OR #Jog_Rev_Req OR #Stop OR NOT #Enable) AND #Abs_Act THEN
       #Abs_Act := FALSE;
   END_IF;
END_REGION

REGION Network 25: Set Request Relative move to Drive (REGISTER 10)
   RUNG wire#powerrail
      Contact( #Start_OS )
      I_Contact( #Abs_Act )
      I_Contact( #Stop_Act )
      I_Contact( #HM_Act )
      { S7_Templates := "SrcType := DInt" } EQ_Contact(in1 := #Move_Type_Loc, in2 := 1)
      S_Coil( #Rel_Act )
   END_RUNG
   RUNG wire#powerrail
      Contact( #Rel_Act )
      P_Trig( #REL_PMem )
      Move(in := #Position_SP, out1 => #Drive_Out.MR)
      { S7_Templates := "time_type := Time" } #REL_Tmr.TOF(pt := T#50ms, et => #_Rel_Tmr_ET)
      Coil( #Drive_Out.Toggle_reg_10 )
   END_RUNG
   RUNG wire#powerrail
      Contact( #MV_Stop_OS )
      wire#w1
      Contact( #Rel_Act )
      R_Coil( #Rel_Act )
   END_RUNG
   RUNG wire#powerrail
      Contact( #Jog_Fwd_Req )
   END_RUNG wire#w1
   RUNG wire#powerrail
      Contact( #Jog_Rev_Req )
   END_RUNG wire#w1
   RUNG wire#powerrail
      Contact( #Stop )
   END_RUNG wire#w1
   RUNG wire#powerrail
      I_Contact( #Enable )
   END_RUNG wire#w1
   // the same network as SCL:
   IF #Start_OS AND NOT #Abs_Act AND NOT #Stop_Act AND NOT #HM_Act AND (#Move_Type_Loc = 1) THEN
       #Rel_Act := TRUE;
   END_IF;
   #_w1 := #Rel_Act AND NOT #REL_PMem;   // rising edge
   #REL_PMem := #Rel_Act;
   IF #_w1 THEN #Drive_Out.MR := #Position_SP; END_IF;
   #REL_Tmr(IN := #_w1, PT := T#50ms, ET => #_Rel_Tmr_ET);   // TOF
   #Drive_Out.Toggle_reg_10 := #REL_Tmr.Q;
   IF (#MV_Stop_OS OR #Jog_Fwd_Req OR #Jog_Rev_Req OR #Stop OR NOT #Enable) AND #Rel_Act THEN
       #Rel_Act := FALSE;
   END_IF;
END_REGION

REGION Network 26: Set Request Homing to Drive (REGISTER 22)
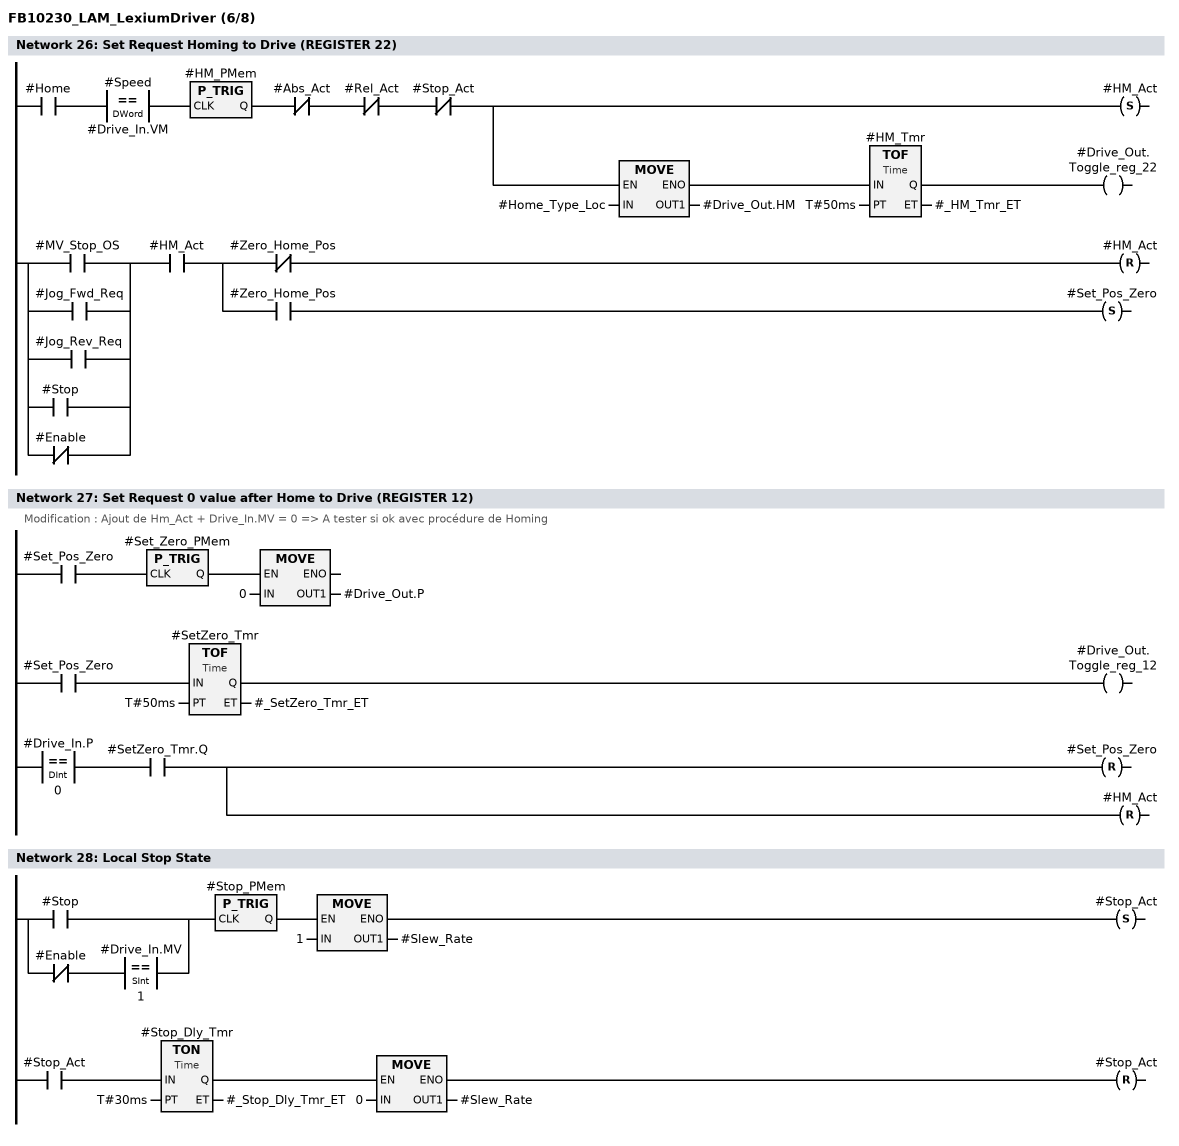
   RUNG wire#powerrail
      Contact( #Home )
      { S7_Templates := "SrcType := DWord" } EQ_Contact(in1 := #Speed, in2 := #Drive_In.VM)
      P_Trig( #HM_PMem )
      I_Contact( #Abs_Act )
      I_Contact( #Rel_Act )
      I_Contact( #Stop_Act )
      wire#w1
      S_Coil( #HM_Act )
   END_RUNG
   RUNG wire#w1
      Move(in := #Home_Type_Loc, out1 => #Drive_Out.HM)
      { S7_Templates := "time_type := Time" } #HM_Tmr.TOF(pt := T#50ms, et => #_HM_Tmr_ET)
      Coil( #Drive_Out.Toggle_reg_22 )
   END_RUNG
   RUNG wire#powerrail
      Contact( #MV_Stop_OS )
      wire#w2
      Contact( #HM_Act )
      wire#w3
      I_Contact( #Zero_Home_Pos )
      R_Coil( #HM_Act )
   END_RUNG
   RUNG wire#powerrail
      Contact( #Jog_Fwd_Req )
   END_RUNG wire#w2
   RUNG wire#powerrail
      Contact( #Jog_Rev_Req )
   END_RUNG wire#w2
   RUNG wire#powerrail
      Contact( #Stop )
   END_RUNG wire#w2
   RUNG wire#powerrail
      I_Contact( #Enable )
   END_RUNG wire#w2
   RUNG wire#w3
      Contact( #Zero_Home_Pos )
      S_Coil( #Set_Pos_Zero )
   END_RUNG
   // the same network as SCL:
   #_w1 := #Home AND (#Speed = #Drive_In.VM);
   #_w2 := #_w1 AND NOT #HM_PMem;   // rising edge
   #HM_PMem := #_w1;
   #_w3 := #_w2 AND NOT #Abs_Act AND NOT #Rel_Act AND NOT #Stop_Act;
   IF #_w3 THEN
       #HM_Act := TRUE;
       #Drive_Out.HM := #Home_Type_Loc;
   END_IF;
   #HM_Tmr(IN := #_w3, PT := T#50ms, ET => #_HM_Tmr_ET);   // TOF
   #Drive_Out.Toggle_reg_22 := #HM_Tmr.Q;
   #_w4 := (#MV_Stop_OS OR #Jog_Fwd_Req OR #Jog_Rev_Req OR #Stop OR NOT #Enable) AND #HM_Act;
   IF #_w4 AND NOT #Zero_Home_Pos THEN #HM_Act := FALSE; END_IF;
   IF #_w4 AND #Zero_Home_Pos THEN #Set_Pos_Zero := TRUE; END_IF;
END_REGION

REGION Network 27: Set Request 0 value after Home to Drive (REGISTER 12)
   // Modification : Ajout de Hm_Act + Drive_In.MV = 0 => A tester si ok avec procédure de Homing
   RUNG wire#powerrail
      Contact( #Set_Pos_Zero )
      P_Trig( #Set_Zero_PMem )
      Move(in := 0, out1 => #Drive_Out.P)
   END_RUNG
   RUNG wire#powerrail
      Contact( #Set_Pos_Zero )
      { S7_Templates := "time_type := Time" } #SetZero_Tmr.TOF(pt := T#50ms, et => #_SetZero_Tmr_ET)
      Coil( #Drive_Out.Toggle_reg_12 )
   END_RUNG
   RUNG wire#powerrail
      { S7_Templates := "SrcType := DInt" } EQ_Contact(in1 := #Drive_In.P, in2 := 0)
      Contact( #SetZero_Tmr.Q )
      wire#w1
      R_Coil( #Set_Pos_Zero )
   END_RUNG
   RUNG wire#w1
      R_Coil( #HM_Act )
   END_RUNG
   // the same network as SCL:
   #_w1 := #Set_Pos_Zero AND NOT #Set_Zero_PMem;   // rising edge
   #Set_Zero_PMem := #Set_Pos_Zero;
   IF #_w1 THEN #Drive_Out.P := 0; END_IF;
   #SetZero_Tmr(IN := #Set_Pos_Zero, PT := T#50ms, ET => #_SetZero_Tmr_ET);   // TOF
   #Drive_Out.Toggle_reg_12 := #SetZero_Tmr.Q;
   IF (#Drive_In.P = 0) AND #SetZero_Tmr.Q THEN
       #Set_Pos_Zero := FALSE;
       #HM_Act := FALSE;
   END_IF;
END_REGION

REGION Network 28: Local Stop State
   RUNG wire#powerrail
      Contact( #Stop )
      wire#w1
      P_Trig( #Stop_PMem )
      Move(in := 1, out1 => #Slew_Rate)
      S_Coil( #Stop_Act )
   END_RUNG
   RUNG wire#powerrail
      I_Contact( #Enable )
      { S7_Templates := "SrcType := SInt" } EQ_Contact(in1 := #Drive_In.MV, in2 := 1)
   END_RUNG wire#w1
   RUNG wire#powerrail
      Contact( #Stop_Act )
      { S7_Templates := "time_type := Time" } #Stop_Dly_Tmr.TON(pt := T#30ms, et => #_Stop_Dly_Tmr_ET)
      Move(in := 0, out1 => #Slew_Rate)
      R_Coil( #Stop_Act )
   END_RUNG
   // the same network as SCL:
   #_w1 := #Stop OR (NOT #Enable AND (#Drive_In.MV = 1));
   #_w2 := #_w1 AND NOT #Stop_PMem;   // rising edge
   #Stop_PMem := #_w1;
   IF #_w2 THEN
       #Slew_Rate := 1;
       #Stop_Act := TRUE;
   END_IF;
   #Stop_Dly_Tmr(IN := #Stop_Act, PT := T#30ms, ET => #_Stop_Dly_Tmr_ET);   // TON
   IF #Stop_Dly_Tmr.Q THEN
       #Slew_Rate := 0;
       #Stop_Act := FALSE;
   END_IF;
END_REGION

REGION Network 29: Output state : Done, error, In Progress
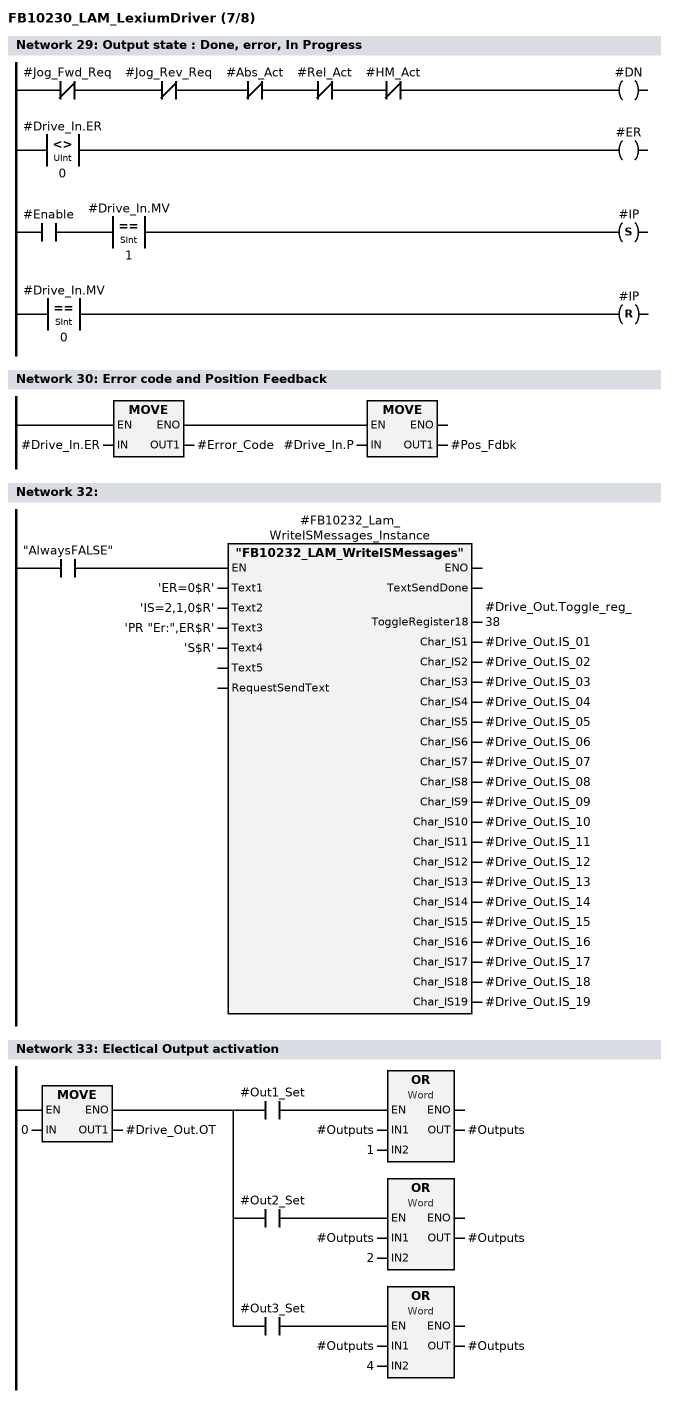
   RUNG wire#powerrail
      I_Contact( #Jog_Fwd_Req )
      I_Contact( #Jog_Rev_Req )
      I_Contact( #Abs_Act )
      I_Contact( #Rel_Act )
      I_Contact( #HM_Act )
      Coil( #DN )
   END_RUNG
   RUNG wire#powerrail
      { S7_Templates := "SrcType := UInt" } NE_Contact(in1 := #Drive_In.ER, in2 := 0)
      Coil( #ER )
   END_RUNG
   RUNG wire#powerrail
      Contact( #Enable )
      { S7_Templates := "SrcType := SInt" } EQ_Contact(in1 := #Drive_In.MV, in2 := 1)
      S_Coil( #IP )
   END_RUNG
   RUNG wire#powerrail
      { S7_Templates := "SrcType := SInt" } EQ_Contact(in1 := #Drive_In.MV, in2 := 0)
      R_Coil( #IP )
   END_RUNG
   // the same network as SCL:
   #DN := NOT #Jog_Fwd_Req AND NOT #Jog_Rev_Req AND NOT #Abs_Act AND NOT #Rel_Act AND NOT #HM_Act;
   #ER := #Drive_In.ER <> 0;
   IF #Enable AND (#Drive_In.MV = 1) THEN #IP := TRUE; END_IF;
   IF #Drive_In.MV = 0 THEN #IP := FALSE; END_IF;
END_REGION

REGION Network 30: Error code and Position Feedback
   RUNG wire#powerrail
      Move(in := #Drive_In.ER, out1 => #Error_Code)
      Move(in := #Drive_In.P, out1 => #Pos_Fdbk)
   END_RUNG
   // the same network as SCL:
   #Error_Code := #Drive_In.ER;
   #Pos_Fdbk := #Drive_In.P;
END_REGION

REGION Network 31 (SCL)
   (*
   IF (NOT #Enable AND (#IS_Config <> #IS_Config_Prev)) OR "FirstScan" THEN
       #IS_PMem := TRUE;
       #Drive_Out.IS_01 := #IS_Config[0];//I
       #Drive_Out.IS_02 := #IS_Config[1];//S
       #Drive_Out.IS_03 := #IS_Config[2];//=
       #Drive_Out.IS_04 := #IS_Config[3];//3
       #Drive_Out.IS_05 := #IS_Config[4];//,
       #Drive_Out.IS_06 := #IS_Config[5];//1
       #Drive_Out.IS_07 := #IS_Config[6];//,
       #Drive_Out.IS_08 := #IS_Config[7];//0
       #Drive_Out.IS_09 := #IS_Config[8];
       #Drive_Out.IS_10 := #IS_Config[9];
       #Drive_Out.IS_11 := #IS_Config[10];
       #Drive_Out.IS_12 := #IS_Config[11];
       #Drive_Out.IS_13 := #IS_Config[12];
       #Drive_Out.IS_14 := #IS_Config[13];
       #Drive_Out.IS_15 := #IS_Config[14];
       #Drive_Out.IS_16 := #IS_Config[15];
       #Drive_Out.IS_17 := #IS_Config[16];
       #Drive_Out.IS_18 := #IS_Config[17];
       #Drive_Out.IS_19 := #IS_Config[18];
       #IS_Config_Prev := #IS_Config;

   END_IF;

   #IS_Config_Tmr(IN := #IS_PMem, PT:=T#50ms);
   //#Drive_Out.Toggle_reg_38 := #IS_Config_Tmr.Q;

   IF #IS_PMem THEN
       #IS_PMem := FALSE;
   END_IF;


   #IS_Config_Prev[0] := '$R';
   #IS_Config_Prev[1] := b#16#1B;
   Chars_TO_Strg(Chars:=#IS_Config_Prev,
                 pChars:=0,
                 Cnt:=2,
                 Strg=>#FB10232_Lam_WriteISMessages_Instance.Text4);
   *)
END_REGION

REGION Network 32
   RUNG wire#powerrail
      Contact( "AlwaysFALSE" )
      #FB10232_Lam_WriteISMessages_Instance(Text1 := 'ER=0$R', Text2 := 'IS=2,1,0$R', Text3 := 'PR "Er:",ER$R', Text4 := 'S$R', Text5 :=, RequestSendText :=, TextSendDone =>, ToggleRegister18 => #Drive_Out.Toggle_reg_38, Char_IS1 => #Drive_Out.IS_01, Char_IS2 => #Drive_Out.IS_02, Char_IS3 => #Drive_Out.IS_03, Char_IS4 => #Drive_Out.IS_04, Char_IS5 => #Drive_Out.IS_05, Char_IS6 => #Drive_Out.IS_06, Char_IS7 => #Drive_Out.IS_07, Char_IS8 => #Drive_Out.IS_08, Char_IS9 => #Drive_Out.IS_09, Char_IS10 => #Drive_Out.IS_10, Char_IS11 => #Drive_Out.IS_11, Char_IS12 => #Drive_Out.IS_12, Char_IS13 => #Drive_Out.IS_13, Char_IS14 => #Drive_Out.IS_14, Char_IS15 => #Drive_Out.IS_15, Char_IS16 => #Drive_Out.IS_16, Char_IS17 => #Drive_Out.IS_17, Char_IS18 => #Drive_Out.IS_18, Char_IS19 => #Drive_Out.IS_19)
   END_RUNG
   // the same network as SCL:
   IF "AlwaysFALSE" THEN
       #FB10232_Lam_WriteISMessages_Instance(Text1 := 'ER=0$R',   // "FB10232_LAM_WriteISMessages"
                               Text2 := 'IS=2,1,0$R',
                               Text3 := 'PR "Er:",ER$R',
                               Text4 := 'S$R',
                               ToggleRegister18 => #Drive_Out.Toggle_reg_38,
                               Char_IS1 => #Drive_Out.IS_01,
                               Char_IS2 => #Drive_Out.IS_02,
                               Char_IS3 => #Drive_Out.IS_03,
                               Char_IS4 => #Drive_Out.IS_04,
                               Char_IS5 => #Drive_Out.IS_05,
                               Char_IS6 => #Drive_Out.IS_06,
                               Char_IS7 => #Drive_Out.IS_07,
                               Char_IS8 => #Drive_Out.IS_08,
                               Char_IS9 => #Drive_Out.IS_09,
                               Char_IS10 => #Drive_Out.IS_10,
                               Char_IS11 => #Drive_Out.IS_11,
                               Char_IS12 => #Drive_Out.IS_12,
                               Char_IS13 => #Drive_Out.IS_13,
                               Char_IS14 => #Drive_Out.IS_14,
                               Char_IS15 => #Drive_Out.IS_15,
                               Char_IS16 => #Drive_Out.IS_16,
                               Char_IS17 => #Drive_Out.IS_17,
                               Char_IS18 => #Drive_Out.IS_18,
                               Char_IS19 => #Drive_Out.IS_19);
   END_IF;
END_REGION

REGION Network 33: Electical Output activation
   #Drive_Out.OT := 0;
   IF #Out1_Set THEN #Outputs := #Outputs OR 1; END_IF;
   IF #Out2_Set THEN #Outputs := #Outputs OR 2; END_IF;
   IF #Out3_Set THEN #Outputs := #Outputs OR 4; END_IF;
END_REGION

REGION Network 34: Set Electrical outputs to Drive
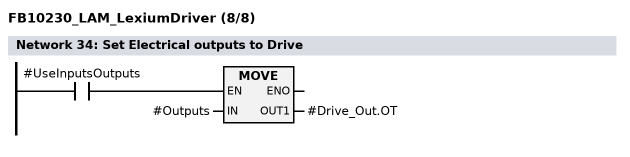
   RUNG wire#powerrail
      Contact( #UseInputsOutputs )
      Move(in := #Outputs, out1 => #Drive_Out.OT)
   END_RUNG
   // the same network as SCL:
   IF #UseInputsOutputs THEN #Drive_Out.OT := #Outputs; END_IF;
END_REGION
END_FUNCTION_BLOCK
